(*
A list implementation for managing `I_Arg`.  
*)
INTERFACE I_MutArgList EXTENDS I_ArgList

(*
Adds, updates, or removes an argument in the list at the specified index.  
Return:
- `Ok` - Upon successfully adding, modifying, or removing an entry.
- `Err.Idx` - When attempting to modify an entry at an out-of-bounds index.
*)
METHOD Set : Result
VAR_INPUT
	iIn		: I_Arg;
	nIndex		: UDINT;
END_VAR
END_METHOD

END_INTERFACE

(* stored: Version 1.1.0.1
   Itf I_MutArgList: Id {6d00e6b1-9212-455b-82a5-6fe0107c2a98}
   Method Set: Id {555f32ab-6a68-4755-ae29-fac819a73af3} *)
